// Mitsubishi GX Works2 project: PLC_GROUP20   PLC: FX3G

// global labels: Global1
VAR_GLOBAL
  SWX10 AT X010 : BOOL;
  Lamp10 AT Y010 : BOOL;
  CurrentOrange AT D1100 : REAL;
END_VAR
VAR_GLOBAL CONSTANT
  Const2 : REAL := 2;
END_VAR
VAR_GLOBAL
  HalfOrange : REAL;
  CurrentMandarine AT D1110 : REAL;
  CurrentPomela AT D1120 : REAL;
  Enough AT M15 : BOOL;
  NotEnoughMaterial AT M145 : BOOL;
  flag1 : BOOL;
  flag2 : BOOL;
  Lamp5 AT Y005 : BOOL;
END_VAR
VAR_GLOBAL CONSTANT
  Const100 : REAL := 100;
END_VAR
VAR_GLOBAL
  TempMovingOrange AT D1140 : REAL;
  CHECK AT D1130 : REAL;
  TempMovingHalf AT D1150 : REAL;
  Switch02 AT X002 : BOOL;
  OrangeWash AT D1160 : REAL;
  MandarineWash AT D1170 : REAL;
  PomelaWash AT D1180 : REAL;
END_VAR
VAR_GLOBAL CONSTANT
  ThreeSec : INT := 30;
END_VAR
VAR_GLOBAL
  Timer3 AT TC4 : BOOL;
  Lamp6 AT Y006 : BOOL;
  AllMoved AT M16 : BOOL;
  Nc AT M145 : BOOL;
  Timer3_out AT TS1 : BOOL;
  Switch01 AT X001 : BOOL;
  Collect_Friut_Stop AT M19 : BOOL;
  Lamp01 AT Y001 : BOOL;
  SqueezeContainer AT D1190 : REAL;
  OrangeWashTemp AT D1250 : REAL;
  PomelaWashTemp AT D1260 : REAL;
  MandarineWashTemp AT D1270 : REAL;
  Lamp27 AT M27 : BOOL;
  SW011 AT X011 : BOOL;
  Lamp28 AT M28 : BOOL;
  Lamp2 AT Y002 : BOOL;
  Blink2 AT M2 : BOOL;
  Blink3 AT M3 : BOOL;
  Blink23 AT M2 : BOOL;
  end_proces AT TS9 : BOOL;
  Blink5 AT M5 : BOOL;
  Lamp3 AT Y003 : BOOL;
  Timer3Sec AT TC1 : BOOL;
  TimerHelper AT TC5 : BOOL;
  Timer3_5_out AT TS5 : BOOL;
  StartQA AT X003 : BOOL;
  FirstTry AT M40 : BOOL;
END_VAR
VAR_GLOBAL CONSTANT
  const_3 : REAL := 5.0;
  Const5 : REAL := 5.0;
END_VAR
VAR_GLOBAL
  NotQualityCheck AT M62 : BOOL;
END_VAR
VAR_GLOBAL CONSTANT
  Const1 : REAL := 1.0;
END_VAR
VAR_GLOBAL
  QualityCheck AT M42 : BOOL;
  FiveSecHelper AT M46 : BOOL;
  Timer5Sec AT TC6 : BOOL;
END_VAR
VAR_GLOBAL CONSTANT
  FiveSec : INT := 50;
END_VAR
VAR_GLOBAL
  Timer5_out AT TS6 : BOOL;
  Lamp4 AT Y004 : BOOL;
END_VAR
VAR_GLOBAL CONSTANT
  Const400 : REAL := 400;
END_VAR
VAR_GLOBAL
  Analog2Input AT D8281 : INT;
  QAValid AT M50 : BOOL;
  JuiceContainer AT D1310 : REAL;
  JuiceIsFull : BOOL;
  SqueezContainerEmpty AT M53 : BOOL;
  Analog2Output AT D8283 : REAL;
END_VAR
VAR_GLOBAL CONSTANT
  const_0 : REAL;
  const_2 : REAL := 2;
END_VAR
VAR_GLOBAL
  Timer8 AT TC8 : BOOL;
  Timer8S AT TS8 : BOOL;
  Timer10 AT TC10 : BOOL;
  Timer10S AT TS10 : BOOL;
  C_2 AT CC1 : BOOL;
END_VAR
VAR_GLOBAL CONSTANT
  Count2 : INT := 2;
END_VAR
VAR_GLOBAL
  BreakSwitchX7 AT X007 : BOOL;
  Counter2 AT CS1 : BOOL;
  flag3 : BOOL;
  Less5 AT M60 : BOOL;
  Greater1 AT M44 : BOOL;
  Analog2Value AT D8283 : REAL;
  Switch06 AT X006 : BOOL;
  Analog1Input AT D8280 : INT;
  Analog1Value AT D8286 : REAL;
  AnalogOutput AT D8282 : REAL;
  Less10 AT M68 : BOOL;
END_VAR
VAR_GLOBAL CONSTANT
  Const_10 : REAL := 10;
END_VAR
VAR_GLOBAL
  MaxFruit AT D1200 : REAL;
  FruitConstraint AT M40 : BOOL;
  AfterSqueezeFlag AT M17 : BOOL;
  AfterWashFlag AT M18 : BOOL;
  Lamp2Flag AT M28 : BOOL;
  CounterFlag AT M28 : BOOL;
END_VAR

// task Task_01 (event TRUE, interval 0, priority 31): POU_01

PROGRAM POU_01
(* structured ladder/FBD written out as ST: instructions are called as NAME(EN, inputs, outputs); _pN, _eN, _tN stand for wires *)
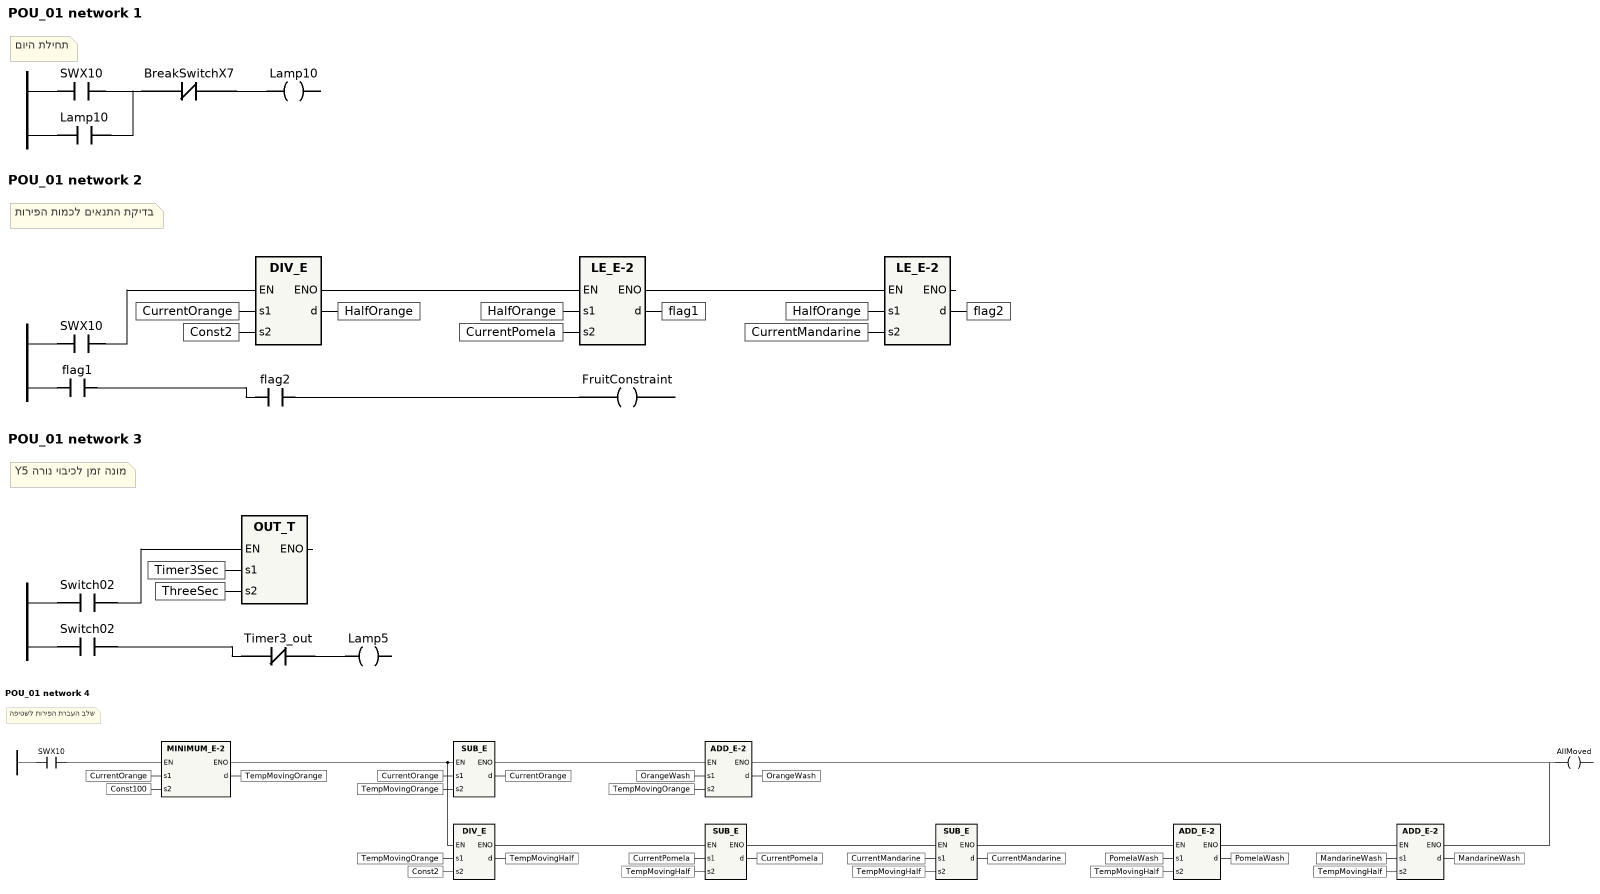
(* network 1 *)
(* תחילת היום *)
Lamp10 := (SWX10 OR Lamp10) AND NOT BreakSwitchX7;
(* network 2 *)
(* בדיקת התנאים לכמות הפירות *)
_e1 := DIV_E(SWX10, CurrentOrange, Const2, HalfOrange);
_e2 := LE_E(_e1, HalfOrange, CurrentPomela, flag1);
LE_E(_e2, HalfOrange, CurrentMandarine, flag2);
FruitConstraint := flag1 AND flag2;
(* network 3 *)
(* מונה זמן לכיבוי נורה Y5 *)
OUT_T(Switch02, Timer3Sec, ThreeSec);
Lamp5 := Switch02 AND NOT Timer3_out;
(* network 4 *)
(* שלב העברת הפירות לשטיפה *)
_e1 := MINIMUM_E(SWX10, CurrentOrange, Const100, TempMovingOrange);
_e2 := SUB_E(_e1, CurrentOrange, TempMovingOrange, CurrentOrange);
_e3 := ADD_E(_e2, OrangeWash, TempMovingOrange, OrangeWash);
_e4 := DIV_E(_e1, TempMovingOrange, Const2, TempMovingHalf);
_e5 := SUB_E(_e4, CurrentPomela, TempMovingHalf, CurrentPomela);
_e6 := SUB_E(_e5, CurrentMandarine, TempMovingHalf, CurrentMandarine);
_e7 := ADD_E(_e6, PomelaWash, TempMovingHalf, PomelaWash);
_e8 := ADD_E(_e7, MandarineWash, TempMovingHalf, MandarineWash);
AllMoved := _e3 OR _e8;
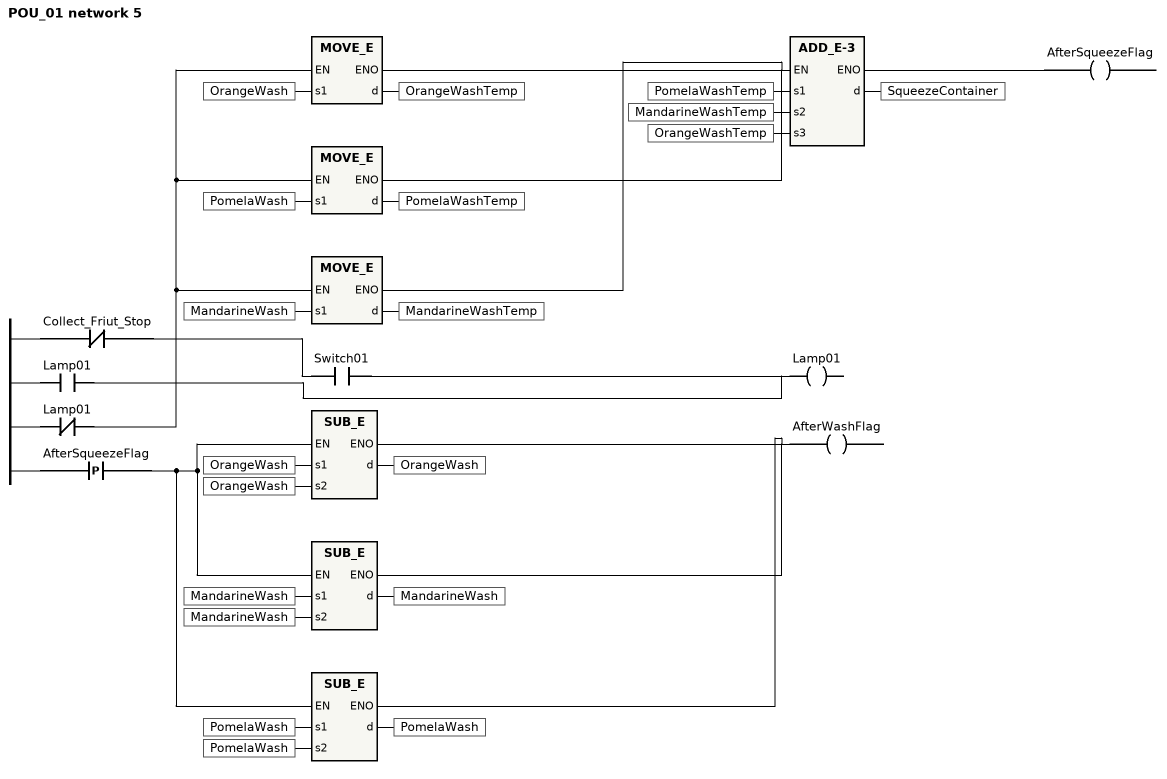
(* network 5 *)
Lamp01 := (NOT Collect_Friut_Stop AND Switch01) OR Lamp01;
_p1 := NOT Lamp01;
_e2 := MOVE_E(_p1, OrangeWash, OrangeWashTemp);
_e3 := MOVE_E(_p1, PomelaWash, PomelaWashTemp);
_e4 := MOVE_E(_p1, MandarineWash, MandarineWashTemp);
_e5 := ADD_E(_e2 OR _e3 OR _e4, PomelaWashTemp, MandarineWashTemp, OrangeWashTemp, SqueezeContainer);
AfterSqueezeFlag := _e5;
_p6 := LDP(TRUE, AfterSqueezeFlag);
_e7 := SUB_E(_p6, OrangeWash, OrangeWash, OrangeWash);
_e8 := SUB_E(_p6, MandarineWash, MandarineWash, MandarineWash);
_e9 := SUB_E(_p6, PomelaWash, PomelaWash, PomelaWash);
AfterWashFlag := _e7 OR _e8 OR _e9;
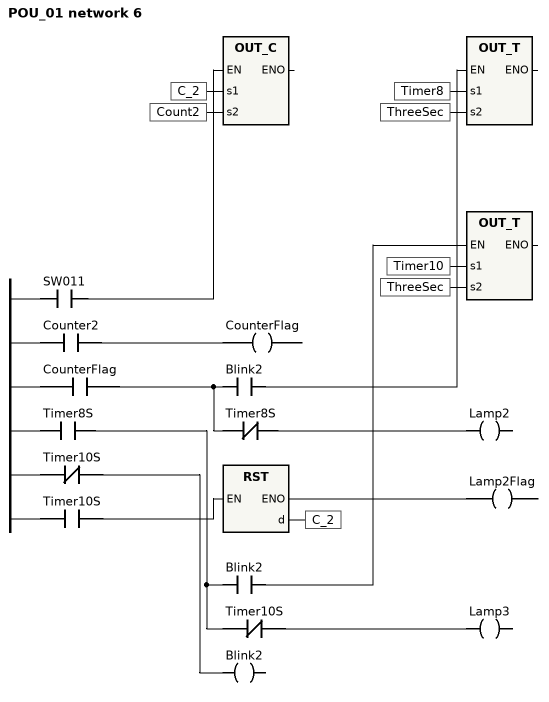
(* network 6 *)
OUT_C(SW011, C_2, Count2);
CounterFlag := Counter2;
OUT_T(CounterFlag AND Blink2, Timer8, ThreeSec);
Lamp2 := CounterFlag AND NOT Timer8S;
OUT_T(Timer8S AND Blink2, Timer10, ThreeSec);
Lamp3 := Timer8S AND NOT Timer10S;
Blink2 := NOT Timer10S;
_e1 := RST(Timer10S, C_2);
Lamp2Flag := _e1;
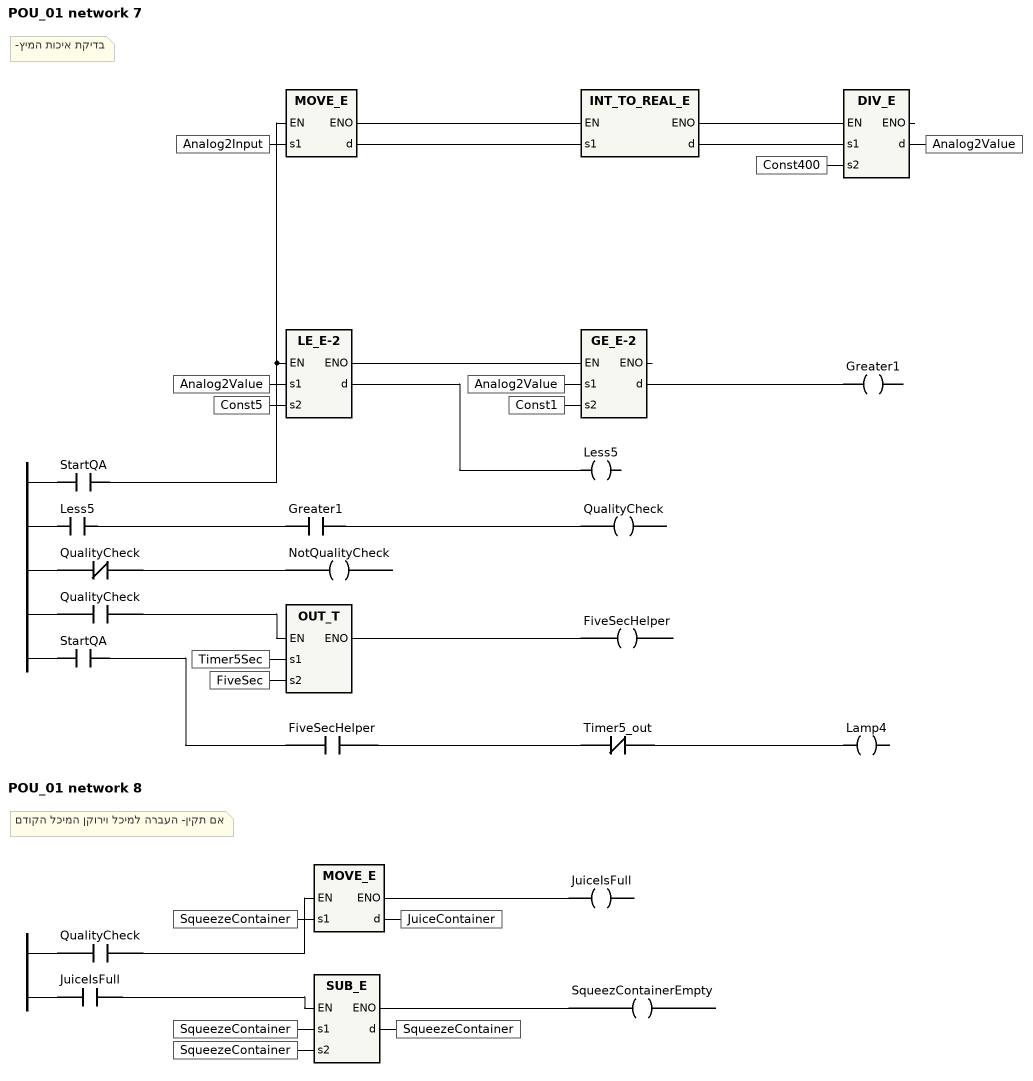
(* network 7 *)
(* בדיקת איכות המיץ- *)
_e2 := MOVE_E(StartQA, Analog2Input, _t1);
_e4 := INT_TO_REAL_E(_e2, _t1, _t3);
DIV_E(_e4, _t3, Const400, Analog2Value);
_e6 := LE_E(StartQA, Analog2Value, Const5, _t5);
GE_E(_e6, Analog2Value, Const1, _t7);
Less5 := _t5;
Greater1 := _t7;
QualityCheck := Less5 AND Greater1;
NotQualityCheck := NOT QualityCheck;
_e8 := OUT_T(QualityCheck, Timer5Sec, FiveSec);
FiveSecHelper := _e8;
Lamp4 := StartQA AND FiveSecHelper AND NOT Timer5_out;
(* network 8 *)
(* אם תקין- העברה למיכל וירוקן המיכל הקודם *)
_e1 := MOVE_E(QualityCheck, SqueezeContainer, JuiceContainer);
JuiceIsFull := _e1;
_e2 := SUB_E(JuiceIsFull, SqueezeContainer, SqueezeContainer, SqueezeContainer);
SqueezContainerEmpty := _e2;
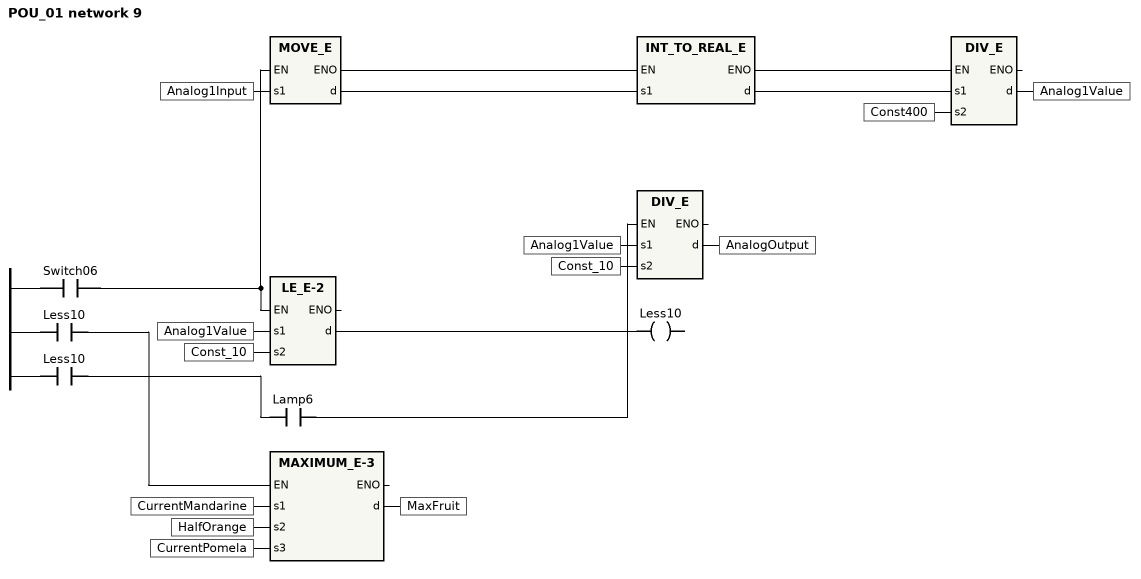
(* network 9 *)
_e2 := MOVE_E(Switch06, Analog1Input, _t1);
_e4 := INT_TO_REAL_E(_e2, _t1, _t3);
DIV_E(_e4, _t3, Const400, Analog1Value);
LE_E(Switch06, Analog1Value, Const_10, _t5);
Less10 := _t5;
MAXIMUM_E(Less10, CurrentMandarine, HalfOrange, CurrentPomela, MaxFruit);
DIV_E(Less10 AND Lamp6, Analog1Value, Const_10, AnalogOutput);
END_PROGRAM
